% RSLogix 500 project P3.RSS, saved by version 8.30.00.16 %
PROJECT "UNTITLED"    % processor: Bul.1763 MicroLogix 1100 Series B %

PROGRAM FILES
  LAD 2   9 rungs

DATA FILES
  O0 OUTPUT  4 elements
  I1 INPUT  6 elements
  S2 STATUS  66 elements
  B3 BINARY  1 elements
  T4 TIMER  1 elements
  C5 COUNTER  1 elements
  R6 CONTROL  1 elements
  N7 INTEGER  4 elements
  F8 FLOAT  1 elements
  ST9 STRINGS  10 elements

LADDER 2
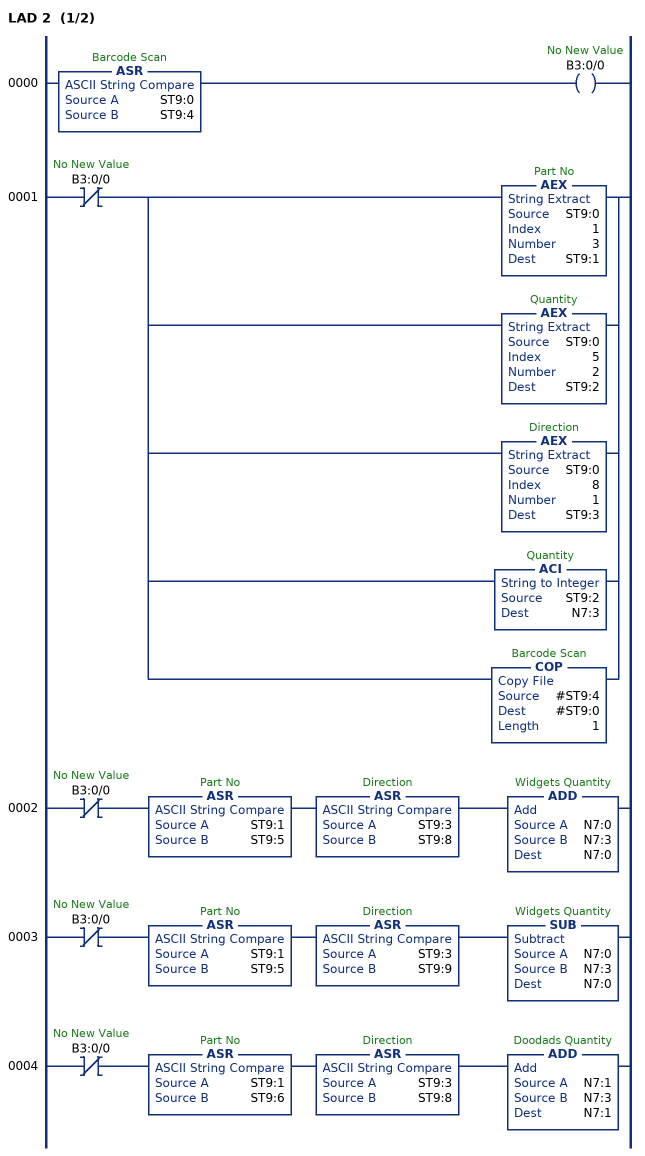
% Rung: 0 %
SOR ASR ST9:0 ST9:4 OTE B3:0/0 EOR
%   ST9:0  "Barcode Scan" %
%   ST9:4  "Empty String (Reset)" %
%   B3:0/0  "No New Value" %
% Rung: 1 %
SOR XIO B3:0/0 BST AEX ST9:0 1 3 ST9:1 NXB AEX ST9:0 5 2 ST9:2 NXB AEX ST9:0 8 1 ST9:3 NXB ACI ST9:2 N7:3 NXB COP #ST9:4 #ST9:0 1 BND EOR
%   B3:0/0  "No New Value" %
%   ST9:0  "Barcode Scan" %
%   ST9:1  "Part No" %
%   ST9:2  "Quantity" %
%   ST9:3  "Direction" %
%   N7:3  "Quantity" %
%   ST9:4  "Empty String (Reset)" %
% Rung: 2 %
SOR XIO B3:0/0 ASR ST9:1 ST9:5 ASR ST9:3 ST9:8 ADD N7:0 N7:3 N7:0 EOR
%   B3:0/0  "No New Value" %
%   ST9:1  "Part No" %
%   ST9:5  "Widgets PN" %
%   ST9:3  "Direction" %
%   ST9:8  "Incoming Direction" %
%   N7:0  "Widgets Quantity" %
%   N7:3  "Quantity" %
% Rung: 3 %
SOR XIO B3:0/0 ASR ST9:1 ST9:5 ASR ST9:3 ST9:9 SUB N7:0 N7:3 N7:0 EOR
%   B3:0/0  "No New Value" %
%   ST9:1  "Part No" %
%   ST9:5  "Widgets PN" %
%   ST9:3  "Direction" %
%   ST9:9  "Outgoing Direction" %
%   N7:0  "Widgets Quantity" %
%   N7:3  "Quantity" %
% Rung: 4 %
SOR XIO B3:0/0 ASR ST9:1 ST9:6 ASR ST9:3 ST9:8 ADD N7:1 N7:3 N7:1 EOR
%   B3:0/0  "No New Value" %
%   ST9:1  "Part No" %
%   ST9:6  "Doodads PN" %
%   ST9:3  "Direction" %
%   ST9:8  "Incoming Direction" %
%   N7:1  "Doodads Quantity" %
%   N7:3  "Quantity" %

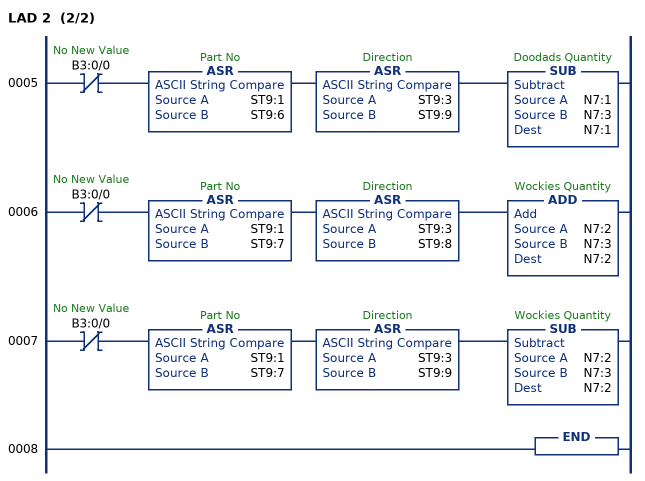
% Rung: 5 %
SOR XIO B3:0/0 ASR ST9:1 ST9:6 ASR ST9:3 ST9:9 SUB N7:1 N7:3 N7:1 EOR
%   B3:0/0  "No New Value" %
%   ST9:1  "Part No" %
%   ST9:6  "Doodads PN" %
%   ST9:3  "Direction" %
%   ST9:9  "Outgoing Direction" %
%   N7:1  "Doodads Quantity" %
%   N7:3  "Quantity" %
% Rung: 6 %
SOR XIO B3:0/0 ASR ST9:1 ST9:7 ASR ST9:3 ST9:8 ADD N7:2 N7:3 N7:2 EOR
%   B3:0/0  "No New Value" %
%   ST9:1  "Part No" %
%   ST9:7  "Wockies PN" %
%   ST9:3  "Direction" %
%   ST9:8  "Incoming Direction" %
%   N7:2  "Wockies Quantity" %
%   N7:3  "Quantity" %
% Rung: 7 %
SOR XIO B3:0/0 ASR ST9:1 ST9:7 ASR ST9:3 ST9:9 SUB N7:2 N7:3 N7:2 EOR
%   B3:0/0  "No New Value" %
%   ST9:1  "Part No" %
%   ST9:7  "Wockies PN" %
%   ST9:3  "Direction" %
%   ST9:9  "Outgoing Direction" %
%   N7:2  "Wockies Quantity" %
%   N7:3  "Quantity" %
% Rung: 8 %
SOR END EOR

DATA TABLE (non-zero values as saved)
DATA ST9
% ST9:1 % "149"
% ST9:2 % "1:"
% ST9:3 % "2"
% ST9:5 % "123"
% ST9:6 % "456"
% ST9:7 % "789"
% ST9:8 % "1"
% ST9:9 % "2"
